N38150 X-5.476 
N38160 X-5.471 
N38170 X-5.465 
N38180 X-5.458 
N38190 X-5.451 
N38200 X-5.443 
N38210 X-5.434 
N38220 X-5.425 
N38230 X-5.416 
N38240 X-5.405 
N38250 X-5.394 
N38260 X-5.383 
N38270 X-5.371 
N38280 X-5.359 
N38290 X-5.346 
N38300 X-5.332 
N38310 X-5.318 
N38320 X-5.303 
N38330 X-5.288 
N38340 X-5.272 
N38350 X-5.256 
N38360 X-5.239 
N38370 X-5.222 
N38380 X-5.204 
N38390 X-5.186 
N38400 X-5.167 
N38410 X-5.147 
N38420 X-5.127 
N38430 X-5.107 
N38440 X-5.086 
N38450 X-5.065 
N38460 X-5.043 
N38470 X-5.021 
N38480 X-4.998 
N38490 X-4.975 
N38500 X-4.952 
N38510 X-4.928 
N38520 X-4.903 
N38530 X-4.878 
N38540 X-4.853 
N38550 X-4.827 
N38560 X-4.801 
N38570 X-4.774 
N38580 X-4.747 
N38590 X-4.72 
N38600 X-4.692 
N38610 X-4.664 
N38620 X-4.635 
N38630 X-4.606 
N38640 X-4.576 
N38650 X-4.547 
N38660 X-4.516 
N38670 X-4.486 
N38680 X-4.455 
N38690 X-4.424 
N38700 X-4.392 
N38710 X-4.36 
N38720 X-4.328 
N38730 X-4.295 
N38740 X-4.262 
N38750 X-4.228 
N38760 X-4.195 
N38770 X-4.161 
N38780 X-4.126 
N38790 X-4.092 
N38800 X-4.022 
N38810 X-3.95 
N38820 X-3.877 
N38830 X-3.804 
N38840 X-3.729 
N38850 X-3.653 
N38860 X-3.576 
N38870 X-3.498 
N38880 X-3.42 
N38890 X-3.34 
N38900 X-3.26 
N38910 X-3.178 
N38920 X-3.096 
N38930 X-3.013 
N38940 X-2.93 
N38950 X-2.846 
N38960 X-2.761 
N38970 X-2.675 
N38980 X-2.589 
N38990 X-2.503 
N39000 X-2.416 
N39010 X-2.329 
N39020 X-2.241 
N39030 X-2.153 
N39040 X-2.065 
N39050 X-1.887 
N39060 X-1.709 
N39070 X-1.351 
N39080 X-1.172 
N39090 X-0.993 
N39100 X-0.815 
N39110 X-0.639 
N39120 X-0.551 
N39130 X-0.463 
N39140 X-0.376 
N39150 X-0.289 
N39160 X-0.203 
N39170 X-0.118 
N39180 X-0.033 
N39190 X0.052 
N39200 X0.136 
N39210 X0.219 
N39220 X0.301 
N39230 X0.383 
N39240 X0.464 
N39250 X0.544 
N39260 X0.623 
N39270 X0.701 
N39280 X0.778 
N39290 X0.854 
N39300 X0.93 
N39310 X1.004 
N39320 X1.077 
N39330 X1.149 
N39340 X1.219 
N39350 X1.254 
N39360 X1.289 
N39370 X1.323 
N39380 X1.357 
N39390 X1.391 
N39400 X1.424 
N39410 X1.457 
N39420 X1.49 
N39430 X1.522 
N39440 X1.554 
N39450 X1.585 
N39460 X1.617 
N39470 X1.648 
N39480 X1.678 
N39490 X1.708 
N39500 X1.738 
N39510 X1.767 
N39520 X1.796 
N39530 X1.825 
N39540 X1.853 
N39550 X1.881 
N39560 X1.908 
N39570 X1.935 
N39580 X1.962 
N39590 X1.988 
N39600 X2.014 
N39610 X2.039 
N39620 X2.064 
N39630 X2.088 
N39640 X2.112 
N39650 X2.136 
N39660 X2.159 
N39670 X2.181 
N39680 X2.203 
N39690 X2.225 
N39700 X2.246 
N39710 X2.267 
N39720 X2.287 
N39730 X2.307 
N39740 X2.326 
N39750 X2.345 
N39760 X2.363 
N39770 X2.381 
N39780 X2.398 
N39790 X2.415 
N39800 X2.431 
N39810 X2.447 
N39820 X2.462 
N39830 X2.476 
N39840 X2.49 
N39850 X2.504 
N39860 X2.517 
N39870 X2.529 
N39880 X2.541 
N39890 X2.552 
N39900 X2.563 
N39910 X2.573 
N39920 X2.583 
N39930 X2.592 
N39940 X2.6 
N39950 X2.608 
N39960 X2.615 
N39970 X2.622 
N39980 X2.628 
N39990 X2.633 
N40000 X2.638 
N40010 X2.642 
N40020 X2.645 
N40030 X2.648 
N40040 X2.65 
N40050 X2.652 
N40060 X2.653 
N40070 X2.653 Y9.259 
N40080 X2.656 Y9.265 
N40090 X2.669 Y9.289 
N40100 X2.682 Y9.313 
N40110 X2.695 Y9.337 
N40120 X2.709 Y9.361 
N40130 X2.723 Y9.384 
N40140 X2.737 Y9.408 
N40150 X2.752 Y9.431 
N40160 X2.767 Y9.453 
N40170 X2.782 Y9.476 
N40180 X2.798 Y9.498 
N40190 X2.814 Y9.52 
N40200 X2.831 Y9.542 
N40210 X2.847 Y9.563 
N40220 X2.864 Y9.584 
N40230 X2.882 Y9.605 
N40240 X2.899 Y9.625 
N40250 X2.917 Y9.646 
N40260 X2.936 Y9.666 
N40270 X2.954 Y9.685 
N40280 X2.973 Y9.705 
N40290 X2.992 Y9.724 
N40300 X3.012 Y9.742 
N40310 X3.031 Y9.761 
N40320 X3.052 Y9.779 
N40330 X3.072 Y9.797 
N40340 X3.092 Y9.814 
N40350 X3.113 Y9.831 
N40360 X3.135 Y9.848 
N40370 X3.156 Y9.865 
N40380 X3.178 Y9.881 
N40390 X3.2 Y9.897 
N40400 X3.222 Y9.912 
N40410 X3.244 Y9.927 
N40420 X3.267 Y9.942 
N40430 X3.29 Y9.956 
N40440 X3.313 Y9.97 
N40450 X3.337 Y9.984 
N40460 X3.36 Y9.997 
N40470 X3.384 Y10.01 
N40480 X3.409 Y10.023 
N40490 X3.433 Y10.035 
N40500 X3.458 Y10.047 
N40510 X3.482 Y10.058 
N40520 X3.507 Y10.069 
N40530 X3.533 Y10.079 
N40540 X3.558 Y10.09 
N40550 X3.584 Y10.099 
N40560 X3.61 Y10.109 
N40570 X3.636 Y10.118 
N40580 X3.662 Y10.126 
N40590 X3.688 Y10.134 
N40600 X3.715 Y10.142 
N40610 X3.742 Y10.149 
N40620 X3.769 Y10.156 
N40630 X3.796 Y10.162 
N40640 X3.824 Y10.168 
N40650 X3.851 Y10.173 
N40660 X3.879 Y10.178 
N40670 X3.907 Y10.183 
N40680 X3.935 Y10.187 
N40690 X3.963 Y10.191 
N40700 X3.991 Y10.194 
N40710 X4.02 Y10.196 
N40720 X4.048 Y10.199 
N40730 X4.077 Y10.2 
N40740 X4.106 Y10.202 
N40750 X4.135 Y10.202 
N40760 X4.164 Y10.203 
N40770 Y10.202 
N40780 Y10.201 
N40790 Y10.199 
N40800 Y10.197 
N40810 Y10.196 
N40820 Y10.195 
N40830 X4.165 Y10.195 
N40840 X4.166 Y10.195 
N40850 X4.168 Y10.195 
N40860 X4.174 Y10.195 
N40870 X4.194 Y10.195 
N40880 X4.235 Y10.193 
N40890 X4.276 Y10.191 
N40900 X4.316 Y10.188 
N40910 X4.356 Y10.184 
N40920 X4.396 Y10.179 
N40930 X4.435 Y10.173 
N40940 X4.475 Y10.166 
N40950 X4.514 Y10.159 
N40960 X4.552 Y10.15 
N40970 X4.591 Y10.141 
N40980 X4.629 Y10.13 
N40990 X4.666 Y10.119 
N41000 X4.703 Y10.107 
N41010 X4.74 Y10.094 
N41020 X4.777 Y10.081 
N41030 X4.813 Y10.066 
N41040 X4.848 Y10.051 
N41050 X4.884 Y10.035 
N41060 X4.918 Y10.018 
N41070 X4.953 Y10 
N41080 X4.987 Y9.982 
N41090 X5.02 Y9.963 
N41100 X5.053 Y9.943 
N41110 X5.086 Y9.923 
N41120 X5.118 Y9.901 
N41130 X5.149 Y9.879 
N41140 X5.18 Y9.857 
N41150 X5.21 Y9.833 
N41160 X5.24 Y9.809 
N41170 X5.27 Y9.785 
N41180 X5.298 Y9.76 
N41190 X5.327 Y9.734 
N41200 X5.354 Y9.707 
N41210 X5.381 Y9.68 
N41220 X5.408 Y9.652 
N41230 X5.433 Y9.624 
N41240 X5.458 Y9.595 
N41250 X5.483 Y9.566 
N41260 X5.507 Y9.536 
N41270 X5.53 Y9.505 
N41280 X5.552 Y9.474 
N41290 X5.574 Y9.443 
N41300 X5.595 Y9.411 
N41310 X5.616 Y9.378 
N41320 X5.635 Y9.345 
N41330 X5.654 Y9.311 
N41340 X5.673 Y9.277 
N41350 X5.69 Y9.243 
N41360 X5.707 Y9.208 
N41370 X5.723 Y9.173 
N41380 X5.738 Y9.137 
N41390 X5.752 Y9.101 
N41400 X5.766 Y9.064 
N41410 X5.778 Y9.027 
N41420 X5.79 Y8.99 
N41430 X5.801 Y8.952 
N41440 X5.811 Y8.914 
N41450 X5.821 Y8.876 
N41460 X5.829 Y8.837 
N41470 X5.836 Y8.798 
N41480 X5.843 Y8.759 
N41490 X5.849 Y8.719 
N41500 X5.854 Y8.679 
N41510 X5.858 Y8.639 
N41520 X5.86 Y8.599 
N41530 X5.862 Y8.558 
N41540 X5.863 Y8.517 
N41550 X5.863 Y8.476 
N41560 X5.863 Y8.435 
N41570 X5.861 Y8.395 
N41580 X5.858 Y8.354 
N41590 X5.854 Y8.314 
N41600 X5.849 Y8.274 
N41610 X5.844 Y8.234 
N41620 X5.837 Y8.195 
N41630 X5.829 Y8.156 
N41640 X5.821 Y8.117 
N41650 X5.812 Y8.079 
N41660 X5.802 Y8.041 
N41670 X5.791 Y8.003 
N41680 X5.779 Y7.966 
N41690 X5.766 Y7.929 
N41700 X5.753 Y7.892 
N41710 X5.739 Y7.856 
N41720 X5.724 Y7.82 
N41730 X5.708 Y7.785 
N41740 X5.691 Y7.75 
N41750 X5.674 Y7.716 
N41760 X5.656 Y7.682 
N41770 X5.637 Y7.648 
N41780 X5.617 Y7.615 
N41790 X5.597 Y7.582 
N41800 X5.576 Y7.55 
N41810 X5.554 Y7.519 
N41820 X5.531 Y7.487 
N41830 X5.508 Y7.457 
N41840 X5.485 Y7.427 
N41850 X5.46 Y7.397 
N41860 X5.435 Y7.369 
N41870 X5.409 Y7.34 
N41880 X5.383 Y7.312 
N41890 X5.356 Y7.285 
N41900 X5.328 Y7.259 
N41910 X5.3 Y7.233 
N41920 X5.272 Y7.207 
N41930 X5.242 Y7.183 
N41940 X5.212 Y7.159 
N41950 X5.182 Y7.135 
N41960 X5.151 Y7.113 
N41970 X5.12 Y7.091 
N41980 X5.088 Y7.07 
N41990 X5.055 Y7.049 
N42000 X5.022 Y7.029 
N42010 X4.989 Y7.01 
N42020 X4.955 Y6.992 
N42030 X4.921 Y6.974 
N42040 X4.886 Y6.957 
N42050 X4.851 Y6.941 
N42060 X4.815 Y6.926 
N42070 X4.779 Y6.911 
N42080 X4.743 Y6.897 
N42090 X4.706 Y6.884 
N42100 X4.669 Y6.872 
N42110 X4.631 Y6.861 
N42120 X4.593 Y6.851 
N42130 X4.555 Y6.841 
N42140 X4.516 Y6.832 
N42150 X4.477 Y6.825 
N42160 X4.438 Y6.818 
N42170 X4.399 Y6.812 
N42180 X4.359 Y6.807 
N42190 X4.319 Y6.803 
N42200 X4.278 Y6.8 
N42210 X4.238 Y6.797 
N42220 X4.197 Y6.796 
N42230 X4.176 Y6.796 
N42240 X4.166 Y6.796 
N42250 X4.164 Y6.796 
N42260 X4.162 Y6.796 
N42270 X4.158 Y6.796 
N42280 X4.129 Y6.796 
N42290 X4.1 Y6.797 
N42300 X4.071 Y6.798 
N42310 X4.042 Y6.8 
N42320 X4.014 Y6.802 
N42330 X3.985 Y6.805 
N42340 X3.957 Y6.808 
N42350 X3.929 Y6.812 
N42360 X3.901 Y6.816 
N42370 X3.873 Y6.821 
N42380 X3.846 Y6.826 
N42390 X3.818 Y6.831 
N42400 X3.791 Y6.837 
N42410 X3.764 Y6.844 
N42420 X3.737 Y6.851 
N42430 X3.71 Y6.858 
N42440 X3.683 Y6.866 
N42450 X3.657 Y6.874 
N42460 X3.631 Y6.882 
N42470 X3.605 Y6.891 
N42480 X3.579 Y6.901 
N42490 X3.553 Y6.911 
N42500 X3.528 Y6.921 
N42510 X3.502 Y6.932 
N42520 X3.477 Y6.943 
N42530 X3.453 Y6.954 
N42540 X3.428 Y6.966 
N42550 X3.404 Y6.978 
N42560 X3.38 Y6.991 
N42570 X3.356 Y7.004 
N42580 X3.332 Y7.017 
N42590 X3.309 Y7.031 
N42600 X3.285 Y7.045 
N42610 X3.263 Y7.059 
N42620 X3.24 Y7.074 
N42630 X3.217 Y7.089 
N42640 X3.195 Y7.105 
N42650 X3.173 Y7.121 
N42660 X3.152 Y7.137 
N42670 X3.13 Y7.153 
N42680 X3.109 Y7.17 
N42690 X3.088 Y7.187 
N42700 X3.068 Y7.205 
N42710 X3.047 Y7.223 
N42720 X3.027 Y7.241 
N42730 X3.008 Y7.259 
N42740 X2.988 Y7.278 
N42750 X2.969 Y7.297 
N42760 X2.95 Y7.317 
N42770 X2.932 Y7.337 
N42780 X2.914 Y7.357 
N42790 X2.896 Y7.377 
N42800 X2.878 Y7.397 
N42810 X2.861 Y7.418 
N42820 X2.844 Y7.44 
N42830 X2.827 Y7.461 
N42840 X2.811 Y7.483 
N42850 X2.795 Y7.505 
N42860 X2.779 Y7.527 
N42870 X2.764 Y7.549 
N42880 X2.749 Y7.572 
N42890 X2.734 Y7.595 
N42900 X2.72 Y7.618 
N42910 X2.706 Y7.642 
N42920 X2.693 Y7.666 
N42930 X2.679 Y7.69 
N42940 X2.666 Y7.714 
N42950 X2.654 Y7.738 
N42960 X2.653 Y7.74 
N42970 X2.652 Y7.74 
N42980 X2.651 
N42990 X2.649 
N43000 X2.646 
N43010 X2.643 
N43020 X2.64 
N43030 X2.635 
N43040 X2.631 
N43050 X2.625 
N43060 X2.619 
N43070 X2.613 
N43080 X2.606 
N43090 X2.598 
N43100 X2.59 
N43110 X2.581 
N43120 X2.572 
N43130 X2.562 
N43140 X2.552 
N43150 X2.541 
N43160 X2.53 
N43170 X2.518 
N43180 X2.505 
N43190 X2.493 
N43200 X2.479 
N43210 X2.465 
N43220 X2.451 
N43230 X2.436 
N43240 X2.421 
N43250 X2.405 
N43260 X2.389 
N43270 X2.372 
N43280 X2.355 
N43290 X2.337 
N43300 X2.319 
N43310 X2.3 
N43320 X2.281 
N43330 X2.262 
N43340 X2.242 
N43350 X2.222 
N43360 X2.201 
N43370 X2.18 
N43380 X2.158 
N43390 X2.136 
N43400 X2.114 
N43410 X2.091 
N43420 X2.067 
N43430 X2.044 
N43440 X2.02 
N43450 X1.995 
N43460 X1.971 
N43470 X1.945 
N43480 X1.92 
N43490 X1.894 
N43500 X1.867 
N43510 X1.841 
N43520 X1.814 
N43530 X1.786 
N43540 X1.759 
N43550 X1.731 
N43560 X1.702 
N43570 X1.673 
N43580 X1.644 
N43590 X1.615 
N43600 X1.585 
N43610 X1.555 
N43620 X1.494 
N43630 X1.432 
N43640 X1.368 
N43650 X1.304 
N43660 X1.238 
N43670 X1.171 
N43680 X1.103 
N43690 X1.034 
N43700 X0.965 
N43710 X0.894 
N43720 X0.822 
N43730 X0.75 
N43740 X0.676 
N43750 X0.602 
N43760 X0.527 
N43770 X0.452 
N43780 X0.375 
N43790 X0.298 
N43800 X0.221 
N43810 X0.143 
N43820 X0.064 
N43830 X-0.015 
N43840 X-0.095 
N43850 X-0.175 
N43860 X-0.256 
N43870 X-0.337 
N43880 X-0.418 
N43890 X-0.581 
N43900 X-0.746 
N43910 X-0.91 
N43920 X-1.241 
N43930 X-1.406 
N43940 X-1.571 
N43950 X-1.734 
N43960 X-1.897 
N43970 X-1.978 
N43980 X-2.058 
N43990 X-2.138 
N44000 X-2.218 
N44010 X-2.297 
N44020 X-2.376 
N44030 X-2.454 
N44040 X-2.531 
N44050 X-2.608 
N44060 X-2.684 
N44070 X-2.76 
N44080 X-2.835 
N44090 X-2.909 
N44100 X-2.982 
N44110 X-3.054 
N44120 X-3.126 
N44130 X-3.196 
N44140 X-3.266 
N44150 X-3.334 
N44160 X-3.402 
N44170 X-3.469 
N44180 X-3.534 
N44190 X-3.599 
N44200 X-3.662 
N44210 X-3.724 
N44220 X-3.754 
N44230 X-3.785 
N44240 X-3.815 
N44250 X-3.844 
N44260 X-3.873 
N44270 X-3.902 
N44280 X-3.931 
N44290 X-3.959 
N44300 X-3.987 
N44310 X-4.015 
N44320 X-4.042 
N44330 X-4.069 
N44340 X-4.095 
N44350 X-4.122 
N44360 X-4.147 
N44370 X-4.173 
N44380 X-4.198 
N44390 X-4.223 
N44400 X-4.247 
N44410 X-4.271 
N44420 X-4.294 
N44430 X-4.317 
N44440 X-4.34 
N44450 X-4.362 
N44460 X-4.384 
N44470 X-4.406 
N44480 X-4.427 
N44490 X-4.447 
N44500 X-4.467 
N44510 X-4.487 
N44520 X-4.506 
N44530 X-4.525 
N44540 X-4.544 
N44550 X-4.562 
N44560 X-4.579 
N44570 X-4.596 
N44580 X-4.613 
N44590 X-4.629 
N44600 X-4.644 
N44610 X-4.66 
N44620 X-4.674 
N44630 X-4.688 
N44640 X-4.702 
N44650 X-4.715 
N44660 X-4.728 
N44670 X-4.74 
N44680 X-4.752 
N44690 X-4.763 
N44700 X-4.773 
N44710 X-4.783 
N44720 X-4.793 
N44730 X-4.802 
N44740 X-4.811 
N44750 X-4.819 
N44760 X-4.826 
N44770 X-4.833 
N44780 X-4.839 
N44790 X-4.845 
N44800 X-4.85 
N44810 X-4.855 
N44820 X-4.859 
N44830 X-4.862 
N44840 X-4.865 
N44850 X-4.867 
N44860 X-4.869 
N44870 X-4.87 
N44880 X-4.871 
N44890 X-4.871 Y7.739 
N44900 X-4.873 Y7.738 
N44910 X-4.875 Y7.736 
N44920 X-4.877 Y7.733 
N44930 X-4.881 Y7.73 
N44940 X-4.885 Y7.726 
N44950 X-4.89 Y7.721 
N44960 X-4.895 Y7.715 
N44970 X-4.901 Y7.709 
N44980 X-4.908 Y7.703 
N44990 X-4.915 Y7.695 
N45000 X-4.923 Y7.687 
N45010 X-4.932 Y7.679 
N45020 X-4.941 Y7.67 
N45030 X-4.951 Y7.66 
N45040 X-4.961 Y7.65 
N45050 X-4.972 Y7.639 
N45060 X-4.984 Y7.627 
N45070 X-4.996 Y7.615 
N45080 X-5.008 Y7.603 
N45090 X-5.021 Y7.59 
N45100 X-5.035 Y7.576 
N45110 X-5.049 Y7.562 
N45120 X-5.063 Y7.548 
N45130 X-5.078 Y7.533 
N45140 X-5.094 Y7.517 
N45150 X-5.11 Y7.501 
N45160 X-5.126 Y7.485 
N45170 X-5.143 Y7.468 
N45180 X-5.16 Y7.451 
N45190 X-5.178 Y7.434 
N45200 X-5.196 Y7.416 
N45210 X-5.214 Y7.397 
N45220 X-5.233 Y7.379 
N45230 X-5.252 Y7.359 
N45240 X-5.272 Y7.34 
N45250 X-5.292 Y7.32 
N45260 X-5.312 Y7.3 
N45270 X-5.333 Y7.28 
N45280 X-5.353 Y7.259 
N45290 X-5.375 Y7.238 
N45300 X-5.396 Y7.216 
N45310 X-5.418 Y7.195 
N45320 X-5.44 Y7.173 
N45330 X-5.462 Y7.151 
N45340 X-5.484 Y7.128 
N45350 X-5.507 Y7.105 
N45360 X-5.553 Y7.059 
N45370 X-5.6 Y7.013 
N45380 X-5.648 Y6.965 
N45390 X-5.696 Y6.917 
N45400 X-5.745 Y6.868 
N45410 X-5.795 Y6.819 
N45420 X-5.844 Y6.769 
N45430 X-5.945 Y6.669 
N45440 X-6.046 Y6.569 
N45450 X-6.146 Y6.468 
N45460 X-6.196 Y6.418 
N45470 X-6.246 Y6.369 
N45480 X-6.296 Y6.32 
N45490 X-6.344 Y6.271 
N45500 X-6.393 Y6.223 
N45510 X-6.44 Y6.175 
N45520 X-6.487 Y6.129 
N45530 X-6.533 Y6.083 
N45540 X-6.556 Y6.06 
N45550 X-6.579 Y6.038 
N45560 X-6.601 Y6.015 
N45570 X-6.623 Y5.994 
N45580 X-6.644 Y5.972 
N45590 X-6.666 Y5.951 
N45600 X-6.687 Y5.93 
N45610 X-6.708 Y5.909 
N45620 X-6.728 Y5.888 
N45630 X-6.748 Y5.868 
N45640 X-6.768 Y5.848 
N45650 X-6.788 Y5.829 
N45660 X-6.807 Y5.81 
N45670 X-6.826 Y5.791 
N45680 X-6.844 Y5.773 
N45690 X-6.862 Y5.755 
N45700 X-6.88 Y5.738 
N45710 X-6.897 Y5.72 
N45720 X-6.914 Y5.704 
N45730 X-6.93 Y5.687 
N45740 X-6.946 Y5.672 
N45750 X-6.961 Y5.656 
N45760 X-6.976 Y5.641 
N45770 X-6.991 Y5.627 
N45780 X-7.005 Y5.613 
N45790 X-7.018 Y5.6 
N45800 X-7.031 Y5.587 
N45810 X-7.044 Y5.574 
N45820 X-7.055 Y5.562 
N45830 X-7.067 Y5.551 
N45840 X-7.078 Y5.54 
N45850 X-7.088 Y5.53 
N45860 X-7.098 Y5.52 
N45870 X-7.107 Y5.511 
N45880 X-7.115 Y5.503 
N45890 X-7.123 Y5.495 
N45900 X-7.13 Y5.488 
N45910 X-7.137 Y5.481 
N45920 X-7.143 Y5.475 
N45930 X-7.148 Y5.47 
N45940 X-7.153 Y5.465 
N45950 X-7.157 Y5.461 
N45960 X-7.161 Y5.457 
N45970 X-7.163 Y5.455 
N45980 X-7.165 Y5.453 
N45990 X-7.166 Y5.452 
N46000 X-7.167 Y5.451 
N46010 X-7.167 Y5.45 
N46020 Y5.448 
N46030 Y5.447 
N46040 Y5.445 
N46050 Y5.443 
N46060 Y5.44 
N46070 Y5.437 
N46080 Y5.434 
N46090 Y5.43 
N46100 Y5.426 
N46110 Y5.422 
N46120 Y5.412 
N46130 Y5.401 
N46140 Y5.389 
N46150 Y5.376 
N46160 Y5.362 
N46170 Y5.347 
N46180 Y5.331 
N46190 Y5.314 
N46200 Y5.296 
N46210 Y5.278 
N46220 Y5.258 
N46230 Y5.238 
N46240 Y5.217 
N46250 Y5.195 
N46260 Y5.173 
N46270 Y5.15 
N46280 Y5.127 
N46290 Y5.103 
N46300 Y5.078 
N46310 Y5.054 
N46320 Y5.003 
N46330 Y4.952 
N46340 Y4.9 
N46350 Y4.847 
N46360 Y4.795 
N46370 Y4.743 
N46380 Y4.692 
N46390 Y4.667 
N46400 Y4.642 
N46410 Y4.617 
N46420 Y4.593 
N46430 Y4.57 
N46440 Y4.546 
N46450 Y4.524 
N46460 Y4.502 
N46470 Y4.481 
N46480 Y4.46 
N46490 Y4.44 
N46500 Y4.421 
N46510 Y4.403 
N46520 Y4.385 
N46530 Y4.369 
N46540 Y4.353 
N46550 Y4.339 
N46560 Y4.325 
N46570 Y4.313 
N46580 Y4.301 
N46590 Y4.291 
N46600 Y4.287 
N46610 Y4.283 
N46620 Y4.279 
N46630 Y4.275 
N46640 Y4.272 
N46650 Y4.269 
N46660 Y4.266 
N46670 Y4.264 
N46680 Y4.262 
N46690 Y4.26 
N46700 Y4.259 
N46710 Y4.258 
N46720 X-7.167 Y4.257 
N46730 X-7.164 Y4.256 
N46740 X-7.139 Y4.243 
N46750 X-7.115 Y4.231 
N46760 X-7.091 Y4.217 
N46770 X-7.067 Y4.204 
N46780 X-7.044 Y4.19 
N46790 X-7.021 Y4.175 
N46800 X-6.998 Y4.161 
N46810 X-6.975 Y4.146 
N46820 X-6.952 Y4.13 
N46830 X-6.93 Y4.115 
N46840 X-6.908 Y4.099 
N46850 X-6.887 Y4.082 
N46860 X-6.865 Y4.066 
N46870 X-6.844 Y4.049 
N46880 X-6.823 Y4.031 
N46890 X-6.803 Y4.014 
N46900 X-6.782 Y3.996 
N46910 X-6.762 Y3.978 
N46920 X-6.743 Y3.959 
N46930 X-6.723 Y3.94 
N46940 X-6.704 Y3.921 
N46950 X-6.685 Y3.902 
N46960 X-6.667 Y3.882 
N46970 X-6.649 Y3.862 
N46980 X-6.631 Y3.842 
N46990 X-6.613 Y3.821 
N47000 X-6.596 Y3.8 
N47010 X-6.579 Y3.779 
N47020 X-6.563 Y3.758 
N47030 X-6.546 Y3.736 
N47040 X-6.531 Y3.714 
N47050 X-6.515 Y3.692 
N47060 X-6.5 Y3.669 
N47070 X-6.485 Y3.647 
N47080 X-6.471 Y3.624 
N47090 X-6.457 Y3.601 
N47100 X-6.443 Y3.577 
N47110 X-6.43 Y3.553 
N47120 X-6.417 Y3.53 
N47130 X-6.404 Y3.505 
N47140 X-6.392 Y3.481 
N47150 X-6.38 Y3.456 
N47160 X-6.369 Y3.432 
N47170 X-6.358 Y3.407 
N47180 X-6.347 Y3.381 
N47190 X-6.337 Y3.356 
N47200 X-6.327 Y3.33 
N47210 X-6.318 Y3.304 
N47220 X-6.309 Y3.278 
N47230 X-6.3 Y3.252 
N47240 X-6.292 Y3.226 
N47250 X-6.284 Y3.199 
N47260 X-6.277 Y3.172 
N47270 X-6.27 Y3.145 
N47280 X-6.264 Y3.118 
N47290 X-6.258 Y3.091 
N47300 X-6.253 Y3.063 
N47310 X-6.248 Y3.036 
N47320 X-6.243 Y3.008 
N47330 X-6.239 Y2.98 
N47340 X-6.235 Y2.952 
N47350 X-6.232 Y2.923 
N47360 X-6.229 Y2.895 
N47370 X-6.227 Y2.866 
N47380 X-6.225 Y2.838 
N47390 X-6.224 Y2.809 
N47400 X-6.223 Y2.78 
N47410 X-6.223 Y2.751 
N47420 X-6.223 Y2.747 
N47430 X-6.223 Y2.742 
N47440 X-6.223 Y2.732 
N47450 X-6.223 Y2.711 
N47460 X-6.224 Y2.67 
N47470 X-6.227 Y2.63 
N47480 X-6.23 Y2.589 
N47490 X-6.234 Y2.549 
N47500 X-6.239 Y2.51 
N47510 X-6.245 Y2.47 
N47520 X-6.252 Y2.431 
N47530 G00 Z5 
N47540 G00 X-9.416 Y8.275 
N47550 G01 Z-5 F254 
N47560 G01 X-9.463 Y8.25 F1200 
N47570 X-9.512 Y8.226 
N47580 X-9.561 Y8.204 
N47590 X-9.611 Y8.183 
N47600 X-9.662 Y8.164 
N47610 X-9.714 Y8.146 
N47620 X-9.767 Y8.13 
N47630 X-9.82 Y8.116 
N47640 X-9.874 Y8.103 
N47650 X-9.928 Y8.092 
N47660 X-9.983 Y8.083 
N47670 X-10.039 Y8.076 
N47680 X-10.095 Y8.07 
N47690 X-10.152 Y8.067 
N47700 X-10.209 Y8.065 
N47710 X-10.267 Y8.065 
N47720 X-10.324 Y8.067 
N47730 X-10.381 Y8.071 
N47740 X-10.437 Y8.077 
N47750 X-10.492 Y8.084 
N47760 X-10.547 Y8.094 
N47770 X-10.602 Y8.105 
N47780 X-10.655 Y8.118 
N47790 X-10.709 Y8.132 
N47800 X-10.761 Y8.148 
N47810 X-10.813 Y8.166 
N47820 X-10.863 Y8.186 
N47830 X-10.914 Y8.207 
N47840 X-10.963 Y8.229 
N47850 X-11.011 Y8.253 
N47860 X-11.059 Y8.279 
N47870 X-11.106 Y8.306 
N47880 X-11.151 Y8.334 
N47890 X-11.196 Y8.364 
N47900 X-11.24 Y8.395 
N47910 X-11.282 Y8.428 
N47920 X-11.324 Y8.462 
N47930 X-11.364 Y8.497 
N47940 X-11.404 Y8.533 
N47950 X-11.442 Y8.571 
N47960 X-11.479 Y8.609 
N47970 X-11.515 Y8.649 
N47980 X-11.55 Y8.69 
N47990 X-11.583 Y8.732 
N48000 X-11.615 Y8.775 
N48010 X-11.646 Y8.819 
N48020 X-11.675 Y8.864 
N48030 X-11.703 Y8.91 
N48040 X-11.729 Y8.957 
N48050 X-11.754 Y9.005 
N48060 X-11.778 Y9.054 
N48070 X-11.8 Y9.104 
N48080 X-11.82 Y9.154 
N48090 X-11.839 Y9.205 
N48100 X-11.856 Y9.257 
N48110 X-11.872 Y9.31 
N48120 X-11.886 Y9.363 
N48130 X-11.898 Y9.417 
N48140 X-11.908 Y9.472 
N48150 X-11.917 Y9.527 
N48160 X-11.924 Y9.583 
N48170 X-11.929 Y9.639 
N48180 X-11.932 Y9.696 
N48190 X-11.933 Y9.753 
N48200 X-11.933 Y9.811 
N48210 X-11.93 Y9.868 
N48220 X-11.926 Y9.924 
N48230 X-11.92 Y9.98 
N48240 X-11.912 Y10.036 
N48250 X-11.902 Y10.091 
N48260 X-11.89 Y10.145 
N48270 X-11.877 Y10.199 
N48280 X-11.862 Y10.252 
N48290 X-11.846 Y10.304 
N48300 X-11.827 Y10.355 
N48310 X-11.808 Y10.406 
N48320 X-11.786 Y10.456 
N48330 X-11.763 Y10.505 
N48340 X-11.739 Y10.553 
N48350 X-11.713 Y10.601 
N48360 X-11.686 Y10.647 
N48370 X-11.657 Y10.692 
N48380 X-11.627 Y10.737 
N48390 X-11.595 Y10.78 
N48400 X-11.562 Y10.823 
N48410 X-11.528 Y10.864 
N48420 X-11.493 Y10.905 
N48430 X-11.456 Y10.944 
N48440 X-11.419 Y10.982 
N48450 X-11.38 Y11.018 
N48460 X-11.34 Y11.054 
N48470 X-11.298 Y11.088 
N48480 X-11.256 Y11.121 
N48490 X-11.213 Y11.153 
N48500 X-11.168 Y11.183 
N48510 X-11.123 Y11.212 
N48520 X-11.077 Y11.24 
N48530 X-11.03 Y11.266 
N48540 X-10.981 Y11.29 
N48550 X-10.932 Y11.314 
N48560 X-10.883 Y11.335 
N48570 X-10.832 Y11.355 
N48580 X-10.781 Y11.374 
N48590 X-10.729 Y11.391 
N48600 X-10.676 Y11.406 
N48610 X-10.622 Y11.419 
N48620 X-10.568 Y11.431 
N48630 X-10.513 Y11.441 
N48640 X-10.458 Y11.449 
N48650 X-10.402 Y11.456 
N48660 X-10.346 Y11.46 
N48670 X-10.289 Y11.463 
N48680 X-10.26 Y11.464 
N48690 X-10.246 Y11.464 
N48700 X-10.238 Y11.464 
N48710 X-10.235 Y11.464 
N48720 X-10.234 
N48730 X-10.233 
N48740 X-10.222 Y11.464 
N48750 X-10.199 Y11.464 
N48760 X-10.152 Y11.461 
N48770 X-10.107 Y11.457 
N48780 X-10.061 Y11.452 
N48790 X-10.016 Y11.446 
N48800 X-9.972 Y11.438 
N48810 X-9.928 Y11.429 
N48820 X-9.884 Y11.419 
N48830 X-9.841 Y11.408 
N48840 X-9.799 Y11.396 
N48850 X-9.757 Y11.384 
N48860 X-9.715 Y11.371 
N48870 X-9.705 Y11.368 
N48880 X-9.7 Y11.367 
N48890 X-9.698 Y11.366 
N48900 X-9.697 Y11.366 
N48910 X-9.697 Y11.367 
N48920 X-9.696 Y11.368 
N48930 X-9.694 Y11.369 
N48940 X-9.692 Y11.371 
N48950 X-9.69 Y11.373 
N48960 X-9.687 Y11.376 
N48970 X-9.684 Y11.379 
N48980 X-9.681 Y11.383 
N48990 X-9.673 Y11.39 
N49000 X-9.664 Y11.4 
N49010 X-9.653 Y11.411 
N49020 X-9.641 Y11.423 
N49030 X-9.627 Y11.436 
N49040 X-9.612 Y11.451 
N49050 X-9.596 Y11.467 
N49060 X-9.578 Y11.485 
N49070 X-9.56 Y11.504 
N49080 X-9.54 Y11.523 
N49090 X-9.519 Y11.544 
N49100 X-9.497 Y11.567 
N49110 X-9.474 Y11.59 
N49120 X-9.449 Y11.614 
N49130 X-9.424 Y11.639 
N49140 X-9.398 Y11.666 
N49150 X-9.37 Y11.693 
N49160 X-9.342 Y11.721 
N49170 X-9.313 Y11.75 
N49180 X-9.283 Y11.78 
N49190 X-9.253 Y11.811 
N49200 X-9.221 Y11.842 
N49210 X-9.189 Y11.874 
N49220 X-9.156 Y11.907 
N49230 X-9.122 Y11.941 
N49240 X-9.088 Y11.975 
N49250 X-9.053 Y12.01 
N49260 X-9.018 Y12.046 
N49270 X-8.982 Y12.082 
N49280 X-8.945 Y12.118 
N49290 X-8.908 Y12.155 
N49300 X-8.871 Y12.193 
N49310 X-8.833 Y12.231 
N49320 X-8.794 Y12.269 
N49330 X-8.717 Y12.346 
N49340 X-8.638 Y12.425 
N49350 X-8.559 Y12.505 
N49360 X-8.238 Y12.825 
N49370 X-8.158 Y12.905 
N49380 X-8.079 Y12.984 
N49390 X-8.002 Y13.062 
N49400 X-7.925 Y13.138 
N49410 X-7.888 Y13.176 
N49420 X-7.85 Y13.213 
N49430 X-7.814 Y13.25 
N49440 X-7.777 Y13.286 
N49450 X-7.742 Y13.322 
N49460 X-7.707 Y13.357 
N49470 X-7.672 Y13.391 
N49480 X-7.638 Y13.425 
N49490 X-7.605 Y13.458 
N49500 X-7.572 Y13.491 
N49510 X-7.541 Y13.523 
N49520 X-7.51 Y13.554 
N49530 X-7.479 Y13.584 
N49540 X-7.45 Y13.613 
N49550 X-7.422 Y13.642 
N49560 X-7.394 Y13.669 
N49570 X-7.367 Y13.696 
N49580 X-7.342 Y13.722 
N49590 X-7.317 Y13.746 
N49600 X-7.293 Y13.77 
N49610 X-7.271 Y13.793 
N49620 X-7.249 Y13.814 
N49630 X-7.229 Y13.834 
N49640 X-7.21 Y13.853 
N49650 X-7.192 Y13.871 
N49660 X-7.175 Y13.888 
N49670 X-7.16 Y13.903 
N49680 X-7.146 Y13.917 
N49690 X-7.133 Y13.93 
N49700 X-7.122 Y13.942 
N49710 X-7.112 Y13.951 
N49720 X-7.103 Y13.96 
N49730 X-7.1 Y13.964 
N49740 X-7.096 Y13.967 
N49750 X-7.093 Y13.97 
N49760 X-7.091 Y13.972 
N49770 X-7.089 Y13.975 
N49780 X-7.087 Y13.976 
N49790 X-7.086 Y13.978 
N49800 X-7.085 Y13.979 
N49810 X-7.084 Y13.979 
N49820 X-7.083 Y13.979 
N49830 X-7.082 
N49840 X-7.081 
N49850 X-7.078 
N49860 X-7.075 
N49870 X-7.072 
N49880 X-7.068 
N49890 X-7.063 
N49900 X-7.057 
N49910 X-7.051 
N49920 X-7.045 
N49930 X-7.038 
N49940 X-7.03 
N49950 X-7.021 
N49960 X-7.012 
N49970 X-7.003 
N49980 X-6.993 
N49990 X-6.982 
N50000 X-6.971 
N50010 X-6.959 
N50020 X-6.946 
N50030 X-6.933 
N50040 X-6.92 
N50050 X-6.906 
N50060 X-6.891 
N50070 X-6.876 
N50080 X-6.86 
N50090 X-6.844 
N50100 X-6.827 
N50110 X-6.809 
N50120 X-6.791 
N50130 X-6.773 
N50140 X-6.754 
N50150 X-6.734 
N50160 X-6.694 
N50170 X-6.651 
N50180 X-6.606 
N50190 X-6.559 
N50200 X-6.51 
N50210 X-6.46 
N50220 X-6.407 
N50230 X-6.352 
N50240 X-6.296 
N50250 X-6.237 
N50260 X-6.177 
N50270 X-6.115 
N50280 X-6.051 
N50290 X-5.986 
N50300 X-5.919 
N50310 X-5.85 
N50320 X-5.779 
N50330 X-5.707 
N50340 X-5.633 
N50350 X-5.557 
N50360 X-5.48 
N50370 X-5.401 
N50380 X-5.321 
N50390 X-5.239 
N50400 X-5.156 
N50410 X-5.072 
N50420 X-4.986 
N50430 X-4.898 
N50440 X-4.81 
N50450 X-4.719 
N50460 X-4.628 
N50470 X-4.535 
N50480 X-4.441 
N50490 X-4.346 
N50500 X-4.25 
N50510 X-4.152 
N50520 X-4.053 
N50530 X-3.953 
N50540 X-3.852 
N50550 X-3.75 
N50560 X-3.647 
N50570 X-3.543 
N50580 X-3.438 
N50590 X-3.332 
N50600 X-3.225 
N50610 X-3.117 
N50620 X-3.008 
N50630 X-2.898 
N50640 X-2.787 
N50650 X-2.676 
N50660 X-2.563 
N50670 X-2.45 
N50680 X-2.337 
N50690 X-2.222 
N50700 X-2.107 
N50710 X-1.991 
N50720 X-1.875 
N50730 X-1.758 
N50740 X-1.64 
N50750 X-1.522 
N50760 X-1.403 
N50770 X-1.164 
N50780 X-0.923 
N50790 X-0.681 
N50800 X-0.437 
N50810 X-0.192 
N50820 X0.054 
N50830 X0.3 
N50840 X0.548 
N50850 X1.538 
N50860 X1.785 
N50870 X2.032 
N50880 X2.277 
N50890 X2.522 
N50900 X2.765 
N50910 X3.006 
N50920 X3.246 
N50930 X3.484 
N50940 X3.602 
N50950 X3.719 
N50960 X3.836 
N50970 X3.953 
N50980 X4.068 
N50990 X4.183 
N51000 X4.298 
N51010 X4.411 
N51020 X4.524 
N51030 X4.636 
N51040 X4.748 
N51050 X4.858 
N51060 X4.968 
N51070 X5.077 
N51080 X5.185 
N51090 X5.292 
N51100 X5.398 
N51110 X5.503 
N51120 X5.607 
N51130 X5.71 
N51140 X5.812 
N51150 X5.912 
N51160 X6.012 
N51170 X6.111 
N51180 X6.208 
N51190 X6.304 
N51200 X6.4 
N51210 X6.493 
N51220 X6.586 
N51230 X6.677 
N51240 X6.767 
N51250 X6.856 
N51260 X6.943 
N51270 X7.029 
N51280 X7.113 
N51290 X7.196 
N51300 X7.278 
N51310 X7.357 
N51320 X7.436 
N51330 X7.513 
N51340 X7.588 
N51350 X7.662 
N51360 X7.734 
N51370 X7.804 
N51380 X7.873 
N51390 X7.94 
N51400 X8.005 
N51410 X8.069 
N51420 X8.131 
N51430 X8.191 
N51440 X8.249 
N51450 X8.305 
N51460 X8.359 
N51470 X8.412 
N51480 X8.462 
N51490 X8.511 
N51500 X8.557 
N51510 X8.602 
N51520 X8.644 
N51530 X8.685 
N51540 X8.704 
N51550 X8.723 
N51560 X8.741 
N51570 X8.759 
N51580 X8.776 
N51590 X8.793 
N51600 X8.809 
N51610 X8.825 
N51620 X8.84 
N51630 X8.855 
N51640 X8.869 
N51650 X8.882 
N51660 X8.895 
N51670 X8.907 
N51680 X8.919 
N51690 X8.93 
N51700 X8.941 
N51710 X8.95 
N51720 X8.96 
N51730 X8.969 
N51740 X8.977 
N51750 X8.985 
N51760 X8.992 
N51770 X8.998 
N51780 X9.004 
N51790 X9.009 
N51800 X9.014 
N51810 X9.018 
N51820 X9.021 
N51830 X9.024 
N51840 X9.026 
N51850 X9.028 
N51860 X9.029 Y13.979 
N51870 X9.03 Y13.978 
N51880 X9.032 Y13.976 
N51890 X9.035 Y13.973 
N51900 X9.039 Y13.969 
N51910 X9.043 Y13.965 
N51920 X9.048 Y13.96 
N51930 X9.054 Y13.954 
N51940 X9.061 Y13.947 
N51950 X9.068 Y13.94 
N51960 X9.077 Y13.932 
N51970 X9.085 Y13.923 
N51980 X9.095 Y13.913 
N51990 X9.105 Y13.903 
N52000 X9.116 Y13.892 
N52010 X9.128 Y13.88 
N52020 X9.14 Y13.868 
N52030 X9.153 Y13.855 
N52040 X9.167 Y13.841 
N52050 X9.181 Y13.827 
N52060 X9.196 Y13.812 
N52070 X9.212 Y13.796 
N52080 X9.228 Y13.78 
N52090 X9.245 Y13.763 
N52100 X9.263 Y13.745 
N52110 X9.281 Y13.727 
N52120 X9.3 Y13.709 
N52130 X9.319 Y13.689 
N52140 X9.339 Y13.669 
N52150 X9.359 Y13.649 
N52160 X9.38 Y13.628 
N52170 X9.402 Y13.606 
N52180 X9.424 Y13.584 
N52190 X9.447 Y13.562 
N52200 X9.47 Y13.538 
N52210 X9.494 Y13.515 
N52220 X9.518 Y13.49 
N52230 X9.543 Y13.466 
N52240 X9.568 Y13.44 
N52250 X9.593 Y13.415 
N52260 X9.62 Y13.388 
N52270 X9.646 Y13.362 
N52280 X9.674 Y13.335 
N52290 X9.701 Y13.307 
N52300 X9.729 Y13.279 
N52310 X9.758 Y13.25 
N52320 X9.787 Y13.222 
N52330 X9.816 Y13.192 
N52340 X9.846 Y13.162 
N52350 X9.876 Y13.132 
N52360 X9.906 Y13.102 
N52370 X9.937 Y13.071 
N52380 X9.969 Y13.039 
N52390 X10.032 Y12.976 
N52400 X10.098 Y12.91 
N52410 X10.164 Y12.844 
N52420 X10.232 Y12.776 
N52430 X10.301 Y12.707 
N52440 X10.371 Y12.637 
N52450 X10.443 Y12.566 
N52460 X10.515 Y12.493 
N52470 X10.588 Y12.42 
N52480 X10.662 Y12.346 
N52490 X10.737 Y12.271 
N52500 X10.813 Y12.195 
N52510 X10.889 Y12.119 
N52520 X10.966 Y12.042 
N52530 X11.044 Y11.964 
N52540 X11.122 Y11.886 
N52550 X11.201 Y11.808 
N52560 X11.359 Y11.65 
N52570 X11.677 Y11.332 
N52580 X11.835 Y11.173 
N52590 X11.994 Y11.014 
N52600 X12.072 Y10.936 
N52610 X12.151 Y10.858 
N52620 X12.228 Y10.78 
N52630 X12.306 Y10.702 
N52640 X12.382 Y10.626 
N52650 X12.458 Y10.55 
N52660 X12.534 Y10.474 
N52670 X12.608 Y10.4 
N52680 X12.682 Y10.326 
N52690 X12.755 Y10.253 
N52700 X12.827 Y10.182 
N52710 X12.897 Y10.111 
N52720 X12.967 Y10.041 
N52730 X13.035 Y9.973 
N52740 X13.103 Y9.906 
N52750 X13.168 Y9.84 
N52760 X13.233 Y9.775 
N52770 X13.265 Y9.744 
N52780 X13.296 Y9.712 
N52790 X13.327 Y9.681 
N52800 X13.357 Y9.651 
N52810 X13.387 Y9.621 
N52820 X13.417 Y9.591 
N52830 X13.447 Y9.562 
N52840 X13.475 Y9.533 
N52850 X13.504 Y9.504 
N52860 X13.532 Y9.476 
N52870 X13.56 Y9.449 
N52880 X13.587 Y9.421 
N52890 X13.613 Y9.395 
N52900 X13.639 Y9.369 
N52910 X13.665 Y9.343 
N52920 X13.69 Y9.318 
N52930 X13.715 Y9.293 
N52940 X13.739 Y9.269 
N52950 X13.763 Y9.245 
N52960 X13.786 Y9.222 
N52970 X13.809 Y9.199 
N52980 X13.831 Y9.177 
N52990 X13.853 Y9.156 
N53000 X13.874 Y9.135 
N53010 X13.894 Y9.114 
N53020 X13.914 Y9.094 
N53030 X13.933 Y9.075 
N53040 X13.952 Y9.056 
N53050 X13.97 Y9.038 
N53060 X13.987 Y9.021 
N53070 X14.004 Y9.004 
N53080 X14.02 Y8.988 
N53090 X14.036 Y8.972 
N53100 X14.051 Y8.957 
N53110 X14.065 Y8.943 
N53120 X14.079 Y8.929 
N53130 X14.092 Y8.916 
N53140 X14.104 Y8.904 
N53150 X14.116 Y8.892 
N53160 X14.127 Y8.881 
N53170 X14.137 Y8.871 
N53180 X14.147 Y8.861 
N53190 X14.156 Y8.853 
N53200 X14.164 Y8.844 
N53210 X14.171 Y8.837 
N53220 X14.178 Y8.83 
N53230 X14.184 Y8.825 
N53240 X14.189 Y8.819 
N53250 X14.193 Y8.815 
N53260 X14.197 Y8.811 
N53270 X14.199 Y8.809 
N53280 X14.201 Y8.807 
N53290 X14.203 Y8.805 
N53300 X14.204 Y8.805 
N53310 X14.207 
N53320 X14.214 
N53330 X14.217 
N53340 X14.218 
N53350 X14.218 Y8.804 
N53360 Y8.802 
N53370 Y8.798 
N53380 Y8.793 
N53390 Y8.786 
N53400 Y8.778 
N53410 Y8.769 
N53420 Y8.757 
N53430 Y8.745 
N53440 Y8.731 
N53450 Y8.716 
N53460 Y8.699 
N53470 Y8.681 
N53480 Y8.662 
N53490 Y8.641 
N53500 Y8.619 
N53510 Y8.596 
N53520 Y8.571 
N53530 Y8.545 
N53540 Y8.518 
N53550 Y8.49 
N53560 Y8.46 
N53570 Y8.43 
N53580 Y8.398 
N53590 Y8.365 
N53600 Y8.33 
N53610 Y8.295 
N53620 Y8.259 
N53630 Y8.221 
N53640 Y8.182 
N53650 Y8.143 
N53660 Y8.102 
N53670 Y8.06 
N53680 Y8.017 
N53690 Y7.973 
N53700 Y7.928 
N53710 Y7.883 
N53720 Y7.836 
N53730 Y7.788 
N53740 Y7.739 
N53750 Y7.69 
N53760 Y7.639 
N53770 Y7.588 
N53780 Y7.536 
N53790 Y7.483 
N53800 Y7.429 
N53810 Y7.374 
N53820 Y7.319 
N53830 Y7.262 
N53840 Y7.205 
N53850 Y7.147 
N53860 Y7.089 
N53870 Y7.029 
N53880 Y6.969 
N53890 Y6.909 
N53900 Y6.847 
N53910 Y6.785 
N53920 Y6.723 
N53930 Y6.659 
N53940 Y6.595 
N53950 Y6.531 
N53960 Y6.466 
N53970 Y6.4 
N53980 Y6.334 
N53990 Y6.267 
N54000 Y6.132 
N54010 Y5.995 
N54020 Y5.857 
N54030 Y5.716 
N54040 Y5.574 
N54050 Y5.431 
N54060 Y5.286 
N54070 Y5.14 
N54080 Y4.993 
N54090 Y4.845 
N54100 Y4.697 
N54110 Y4.547 
N54120 Y4.247 
N54130 Y3.644 
N54140 Y3.343 
N54150 Y3.194 
N54160 Y3.045 
N54170 Y2.896 
N54180 Y2.749 
N54190 Y2.602 
N54200 Y2.457 
N54210 Y2.313 
N54220 Y2.17 
N54230 Y2.029 
N54240 Y1.889 
N54250 Y1.751 
N54260 Y1.615 
N54270 Y1.481 
N54280 Y1.414 
N54290 Y1.349 
N54300 Y1.283 
N54310 Y1.219 
N54320 Y1.155 
N54330 Y1.091 
N54340 Y1.029 
N54350 Y0.967 
N54360 Y0.905 
N54370 Y0.844 
N54380 Y0.784 
N54390 Y0.725 
N54400 Y0.666 
N54410 Y0.608 
N54420 Y0.551 
N54430 Y0.495 
N54440 Y0.439 
N54450 Y0.384 
N54460 Y0.33 
N54470 Y0.277 
N54480 Y0.224 
N54490 Y0.173 
N54500 Y0.122 
N54510 Y0.073 
N54520 Y0.024 
N54530 Y-0.024 
N54540 Y-0.071 
N54550 Y-0.117 
N54560 Y-0.162 
N54570 Y-0.206 
N54580 Y-0.249 
N54590 Y-0.291 
N54600 Y-0.332 
N54610 Y-0.372 
N54620 Y-0.411 
N54630 Y-0.448 
N54640 Y-0.485 
N54650 Y-0.52 
N54660 Y-0.555 
N54670 Y-0.588 
N54680 Y-0.62 
N54690 Y-0.651 
N54700 Y-0.681 
N54710 Y-0.709 
N54720 Y-0.736 
N54730 Y-0.762 
N54740 Y-0.787 
N54750 Y-0.811 
N54760 Y-0.833 
N54770 Y-0.854 
N54780 Y-0.873 
N54790 Y-0.892 
N54800 Y-0.908 
N54810 Y-0.924 
N54820 Y-0.938 
N54830 Y-0.951 
N54840 Y-0.962 
N54850 Y-0.972 
N54860 Y-0.98 
N54870 Y-0.987 
N54880 Y-0.993 
N54890 Y-0.997 
N54900 Y-0.999 
N54910 Y-1 
N54920 X14.217 Y-1.001 
N54930 X14.216 Y-1.002 
N54940 X14.214 Y-1.004 
N54950 X14.212 Y-1.006 
N54960 X14.209 Y-1.009 
N54970 X14.206 Y-1.012 
N54980 X14.202 Y-1.016 
N54990 X14.198 Y-1.02 
N55000 X14.193 Y-1.025 
N55010 X14.188 Y-1.031 
N55020 X14.182 Y-1.036 
N55030 X14.176 Y-1.042 
N55040 X14.169 Y-1.049 
N55050 X14.162 Y-1.056 
N55060 X14.154 Y-1.064 
N55070 X14.146 Y-1.072 
N55080 X14.138 Y-1.08 
N55090 X14.129 Y-1.089 
N55100 X14.12 Y-1.098 
N55110 X14.11 Y-1.108 
N55120 X14.1 Y-1.118 
N55130 X14.089 Y-1.129 
N55140 X14.078 Y-1.14 
N55150 X14.067 Y-1.151 
N55160 X14.055 Y-1.163 
N55170 X14.043 Y-1.175 
N55180 X14.03 Y-1.188 
N55190 X14.017 Y-1.201 
N55200 X14.004 Y-1.214 
N55210 X13.976 Y-1.242 
N55220 X13.947 Y-1.271 
N55230 X13.916 Y-1.302 
N55240 X13.884 Y-1.334 
N55250 X13.851 Y-1.367 
N55260 X13.817 Y-1.401 
N55270 X13.781 Y-1.437 
N55280 X13.744 Y-1.474 
N55290 X13.706 Y-1.512 
N55300 X13.667 Y-1.551 
N55310 X13.627 Y-1.591 
N55320 X13.586 Y-1.633 
N55330 X13.544 Y-1.675 
N55340 X13.501 Y-1.718 
N55350 X13.457 Y-1.762 
N55360 X13.412 Y-1.806 
N55370 X13.366 Y-1.852 
N55380 X13.32 Y-1.898 
N55390 X13.273 Y-1.945 
N55400 X13.226 Y-1.992 
N55410 X13.178 Y-2.041 
N55420 X13.129 Y-2.089 
N55430 X13.08 Y-2.139 
N55440 X13.03 Y-2.188 
N55450 X12.98 Y-2.238 
N55460 X12.929 Y-2.289 
N55470 X12.827 Y-2.391 
N55480 X12.724 Y-2.494 
N55490 X12.516 Y-2.702 
N55500 X12.412 Y-2.806 
N55510 X12.309 Y-2.91 
N55520 X12.206 Y-3.013 
N55530 X12.104 Y-3.114 
N55540 X12.053 Y-3.165 
N55550 X12.003 Y-3.215 
N55560 X11.954 Y-3.264 
N55570 X11.905 Y-3.313 
N55580 X11.856 Y-3.362 
N55590 X11.808 Y-3.41 
N55600 X11.761 Y-3.457 
N55610 X11.714 Y-3.504 
N55620 X11.668 Y-3.55 
N55630 X11.623 Y-3.595 
N55640 X11.579 Y-3.639 
N55650 X11.535 Y-3.683 
N55660 X11.493 Y-3.726 
N55670 X11.451 Y-3.767 
N55680 X11.41 Y-3.808 
N55690 X11.37 Y-3.848 
N55700 X11.332 Y-3.887 
N55710 X11.294 Y-3.924 
N55720 X11.258 Y-3.961 
N55730 X11.222 Y-3.996 
N55740 X11.188 Y-4.03 
N55750 X11.155 Y-4.063 
N55760 X11.124 Y-4.094 
N55770 X11.094 Y-4.124 
N55780 X11.065 Y-4.153 
N55790 X11.038 Y-4.18 
N55800 X11.025 Y-4.193 
N55810 X11.012 Y-4.206 
N55820 X11 Y-4.218 
N55830 X10.988 Y-4.23 
N55840 X10.977 Y-4.241 
N55850 X10.966 Y-4.252 
N55860 X10.955 Y-4.263 
N55870 X10.945 Y-4.273 
N55880 X10.935 Y-4.283 
N55890 X10.925 Y-4.293 
N55900 X10.916 Y-4.302 
N55910 X10.908 Y-4.31 
N55920 X10.9 Y-4.318 
N55930 X10.892 Y-4.326 
N55940 X10.885 Y-4.333 
N55950 X10.878 Y-4.34 
N55960 X10.872 Y-4.346 
N55970 X10.866 Y-4.352 
N55980 X10.861 Y-4.358 
N55990 X10.856 Y-4.363 
N56000 X10.851 Y-4.367 
N56010 X10.847 Y-4.371 
N56020 X10.844 Y-4.374 
N56030 X10.841 Y-4.377 
N56040 X10.839 Y-4.38 
N56050 X10.837 Y-4.382 
N56060 X10.835 Y-4.383 
N56070 X10.834 Y-4.384 
N56080 X10.834 Y-4.385 
N56090 X10.835 Y-4.386 
N56100 X10.836 Y-4.392 
N56110 X10.84 Y-4.402 
N56120 X10.852 Y-4.445 
N56130 X10.864 Y-4.488 
N56140 X10.875 Y-4.531 
N56150 X10.885 Y-4.574 
N56160 X10.894 Y-4.618 
N56170 X10.902 Y-4.661 
N56180 X10.909 Y-4.705 
N56190 X10.915 Y-4.749 
N56200 X10.919 Y-4.794 
N56210 X10.922 Y-4.839 
N56220 X10.924 Y-4.885 
N56230 X10.925 Y-4.908 
N56240 X10.925 Y-4.92 
N56250 X10.925 Y-4.921 
N56260 X10.925 Y-4.925 
N56270 X10.925 Y-4.932 
N56280 X10.924 Y-4.946 
N56290 X10.924 Y-4.975 
N56300 X10.921 Y-5.032 
N56310 X10.916 Y-5.089 
N56320 X10.91 Y-5.144 
N56330 X10.902 Y-5.2 
N56340 X10.892 Y-5.255 
N56350 X10.88 Y-5.309 
N56360 X10.866 Y-5.362 
N56370 X10.851 Y-5.415 
N56380 X10.834 Y-5.467 
N56390 X10.816 Y-5.519 
N56400 X10.796 Y-5.569 
N56410 X10.774 Y-5.619 
N56420 X10.751 Y-5.668 
N56430 X10.726 Y-5.716 
N56440 X10.7 Y-5.763 
N56450 X10.673 Y-5.81 
N56460 X10.644 Y-5.855 
N56470 X10.614 Y-5.899 
N56480 X10.582 Y-5.943 
N56490 X10.549 Y-5.985 
N56500 X10.515 Y-6.026 
N56510 X10.479 Y-6.066 
N56520 X10.442 Y-6.105 
N56530 X10.404 Y-6.143 
N56540 X10.365 Y-6.18 
N56550 X10.325 Y-6.215 
N56560 X10.284 Y-6.249 
N56570 X10.241 Y-6.282 
N56580 X10.198 Y-6.313 
N56590 X10.153 Y-6.343 
N56600 X10.108 Y-6.372 
N56610 X10.061 Y-6.4 
N56620 X10.014 Y-6.425 
N56630 X9.966 Y-6.45 
N56640 X9.917 Y-6.473 
N56650 X9.867 Y-6.494 
N56660 X9.816 Y-6.514 
N56670 X9.764 Y-6.532 
N56680 X9.712 Y-6.549 
N56690 X9.659 Y-6.564 
N56700 X9.606 Y-6.577 
N56710 X9.551 Y-6.589 
N56720 X9.497 Y-6.598 
N56730 X9.441 Y-6.606 
N56740 X9.385 Y-6.613 
N56750 X9.329 Y-6.617 
N56760 X9.272 Y-6.619 
N56770 X9.214 Y-6.62 
N56780 X9.157 Y-6.619 
N56790 X9.1 Y-6.616 
N56800 X9.044 Y-6.61 
N56810 X8.988 Y-6.604 
N56820 X8.933 Y-6.595 
N56830 X8.878 Y-6.584 
N56840 X8.824 Y-6.572 
N56850 X8.771 Y-6.558 
N56860 X8.718 Y-6.543 
N56870 X8.666 Y-6.525 
N56880 X8.615 Y-6.507 
N56890 X8.564 Y-6.486 
N56900 X8.515 Y-6.464 
N56910 X8.466 Y-6.441 
N56920 X8.418 Y-6.416 
N56930 X8.371 Y-6.389 
N56940 X8.325 Y-6.361 
N56950 X8.28 Y-6.332 
N56960 X8.236 Y-6.301 
N56970 X8.193 Y-6.269 
N56980 X8.151 Y-6.236 
N56990 X8.11 Y-6.202 
N57000 X8.07 Y-6.166 
N57010 X8.031 Y-6.129 
N57020 X7.994 Y-6.09 
N57030 X7.957 Y-6.051 
N57040 X7.922 Y-6.011 
N57050 X7.889 Y-5.969 
N57060 X7.856 Y-5.926 
N57070 X7.825 Y-5.883 
N57080 X7.795 Y-5.838 
N57090 X7.767 Y-5.792 
N57100 X7.74 Y-5.745 
N57110 X7.714 Y-5.698 
N57120 X7.69 Y-5.649 
N57130 X7.667 Y-5.6 
N57140 X7.646 Y-5.55 
N57150 X7.627 Y-5.499 
N57160 X7.609 Y-5.447 
N57170 X7.593 Y-5.395 
N57180 X7.578 Y-5.342 
N57190 X7.566 Y-5.288 
N57200 X7.554 Y-5.234 
N57210 X7.545 Y-5.179 
N57220 X7.537 Y-5.123 
N57230 X7.532 Y-5.067 
N57240 X7.528 Y-5.01 
N57250 X7.526 Y-4.953 
N57260 X7.526 Y-4.896 
N57270 X7.527 Y-4.839 
N57280 X7.531 Y-4.782 
N57290 X7.537 Y-4.726 
N57300 X7.544 Y-4.67 
N57310 X7.553 Y-4.615 
N57320 X7.564 Y-4.56 
N57330 X7.576 Y-4.507 
N57340 X7.591 Y-4.453 
N57350 X7.607 Y-4.401 
N57360 X7.624 Y-4.349 
N57370 X7.644 Y-4.298 
N57380 X7.664 Y-4.248 
N57390 X7.687 Y-4.198 
N57400 X7.711 Y-4.15 
N57410 X7.736 Y-4.102 
N57420 X7.763 Y-4.055 
N57430 X7.791 Y-4.01 
N57440 X7.821 Y-3.965 
N57450 X7.852 Y-3.921 
N57460 X7.884 Y-3.878 
N57470 X7.917 Y-3.836 
N57480 X7.952 Y-3.796 
N57490 X7.988 Y-3.756 
N57500 X8.026 Y-3.718 
N57510 X8.064 Y-3.68 
N57520 X8.104 Y-3.644 
N57530 X8.145 Y-3.61 
N57540 X8.187 Y-3.576 
N57550 X8.23 Y-3.544 
N57560 X8.274 Y-3.513 
N57570 X8.318 Y-3.484 
N57580 X8.364 Y-3.455 
N57590 X8.411 Y-3.429 
N57600 X8.459 Y-3.404 
N57610 X8.508 Y-3.38 
N57620 X8.557 Y-3.358 
N57630 X8.607 Y-3.337 
N57640 X8.659 Y-3.318 
N57650 X8.71 Y-3.301 
N57660 X8.763 Y-3.285 
N57670 X8.816 Y-3.271 
N57680 X8.87 Y-3.258 
N57690 X8.925 Y-3.247 
N57700 X8.98 Y-3.238 
N57710 X9.036 Y-3.231 
N57720 X9.092 Y-3.226 
N57730 X9.149 Y-3.223 
N57740 X9.206 Y-3.221 
N57750 X9.22 Y-3.221 
N57760 X9.224 Y-3.221 
N57770 X9.225 Y-3.221 
N57780 X9.226 
N57790 X9.227 Y-3.221 
N57800 X9.233 Y-3.221 
N57810 X9.256 Y-3.221 
N57820 X9.302 Y-3.223 
N57830 X9.348 Y-3.226 
N57840 X9.393 Y-3.23 
N57850 X9.438 Y-3.236 
N57860 X9.483 Y-3.243 
N57870 X9.527 Y-3.251 
N57880 X9.571 Y-3.26 
N57890 X9.614 Y-3.27 
N57900 X9.656 Y-3.281 
N57910 X9.698 Y-3.292 
N57920 X9.74 Y-3.305 
N57930 X9.76 Y-3.311 
N57940 X9.761 Y-3.311 
N57950 X9.762 Y-3.311 
N57960 X9.763 Y-3.31 
N57970 X9.764 Y-3.308 
N57980 X9.766 Y-3.307 
N57990 X9.769 Y-3.304 
N58000 X9.771 Y-3.302 
N58010 X9.774 Y-3.298 
N58020 X9.778 Y-3.295 
N58030 X9.782 Y-3.291 
N58040 X9.787 Y-3.286 
N58050 X9.791 Y-3.281 
N58060 X9.797 Y-3.276 
N58070 X9.802 Y-3.27 
N58080 X9.808 Y-3.264 
N58090 X9.815 Y-3.258 
N58100 X9.822 Y-3.251 
N58110 X9.829 Y-3.244 
N58120 X9.837 Y-3.236 
N58130 X9.845 Y-3.228 
N58140 X9.862 Y-3.211 
N58150 X9.88 Y-3.193 
N58160 X9.9 Y-3.173 
N58170 X9.921 Y-3.151 
N58180 X9.944 Y-3.129 
N58190 X9.968 Y-3.105 
N58200 X9.993 Y-3.08 
N58210 X10.02 Y-3.053 
N58220 X10.047 Y-3.026 
N58230 X10.076 Y-2.997 
N58240 X10.106 Y-2.967 
N58250 X10.137 Y-2.936 
N58260 X10.168 Y-2.904 
N58270 X10.201 Y-2.872 
N58280 X10.235 Y-2.838 
N58290 X10.27 Y-2.803 
N58300 X10.305 Y-2.767 
N58310 X10.342 Y-2.731 
N58320 X10.379 Y-2.694 
N58330 X10.417 Y-2.656 
N58340 X10.456 Y-2.617 
N58350 X10.495 Y-2.578 
N58360 X10.535 Y-2.537 
N58370 X10.576 Y-2.497 
N58380 X10.617 Y-2.456 
N58390 X10.659 Y-2.414 
N58400 X10.701 Y-2.372 
N58410 X10.744 Y-2.329 
N58420 X10.787 Y-2.286 
N58430 X10.831 Y-2.242 
N58440 X10.919 Y-2.154 
N58450 X11.008 Y-2.065 
N58460 X11.097 Y-1.975 
N58470 X11.188 Y-1.885 
N58480 X11.368 Y-1.705 
N58490 X11.458 Y-1.615 
N58500 X11.547 Y-1.526 
N58510 X11.635 Y-1.438 
N58520 X11.678 Y-1.395 
N58530 X11.721 Y-1.351 
N58540 X11.764 Y-1.309 
N58550 X11.806 Y-1.267 
N58560 X11.848 Y-1.225 
N58570 X11.889 Y-1.184 
N58580 X11.93 Y-1.143 
N58590 X11.97 Y-1.103 
N58600 X12.009 Y-1.064 
N58610 X12.048 Y-1.025 
N58620 X12.086 Y-0.987 
N58630 X12.123 Y-0.95 
N58640 X12.159 Y-0.914 
N58650 X12.195 Y-0.878 
N58660 X12.229 Y-0.843 
N58670 X12.263 Y-0.81 
N58680 X12.296 Y-0.777 
N58690 X12.328 Y-0.745 
N58700 X12.358 Y-0.714 
N58710 X12.388 Y-0.685 
N58720 X12.417 Y-0.656 
N58730 X12.444 Y-0.629 
N58740 X12.471 Y-0.602 
N58750 X12.496 Y-0.577 
N58760 X12.519 Y-0.553 
N58770 X12.542 Y-0.531 
N58780 X12.563 Y-0.51 
N58790 X12.583 Y-0.49 
N58800 X12.601 Y-0.472 
N58810 X12.618 Y-0.455 
N58820 X12.626 Y-0.447 
N58830 X12.634 Y-0.439 
N58840 X12.641 Y-0.432 
N58850 X12.648 Y-0.425 
N58860 X12.654 Y-0.419 
N58870 X12.66 Y-0.413 
N58880 X12.666 Y-0.407 
N58890 X12.671 Y-0.402 
N58900 X12.676 Y-0.397 
N58910 X12.68 Y-0.393 
N58920 X12.684 Y-0.389 
N58930 X12.687 Y-0.385 
N58940 X12.69 Y-0.382 
N58950 X12.693 Y-0.38 
N58960 X12.695 Y-0.377 
N58970 X12.697 Y-0.376 
N58980 X12.699 Y-0.374 
N58990 X12.699 Y-0.373 
N59000 X12.7 Y-0.373 
N59010 Y-0.371 
N59020 Y-0.369 
N59030 Y-0.364 
N59040 Y-0.359 
N59050 Y-0.352 
N59060 Y-0.344 
N59070 Y-0.335 
N59080 Y-0.325 
N59090 Y-0.313 
N59100 Y-0.3 
N59110 Y-0.286 
N59120 Y-0.271 
N59130 Y-0.254 
N59140 Y-0.237 
N59150 Y-0.218 
N59160 Y-0.198 
N59170 Y-0.177 
N59180 Y-0.155 
N59190 Y-0.132 
N59200 Y-0.107 
N59210 Y-0.082 
N59220 Y-0.056 
N59230 Y-0.028 
N59240 Y0 
N59250 Y0.03 
N59260 Y0.06 
N59270 Y0.092 
N59280 Y0.124 
N59290 Y0.158 
N59300 Y0.192 
N59310 Y0.227 
N59320 Y0.263 
N59330 Y0.3 
N59340 Y0.338 
N59350 Y0.377 
N59360 Y0.417 
N59370 Y0.457 
N59380 Y0.499 
N59390 Y0.541 
N59400 Y0.584 
N59410 Y0.628 
N59420 Y0.672 
N59430 Y0.717 
N59440 Y0.764 
N59450 Y0.81 
N59460 Y0.858 
N59470 Y0.906 
N59480 Y0.955 
N59490 Y1.004 
N59500 Y1.055 
N59510 Y1.106 
N59520 Y1.157 
N59530 Y1.209 
N59540 Y1.262 
N59550 Y1.315 
N59560 Y1.369 
N59570 Y1.424 
N59580 Y1.479 
N59590 Y1.534 
N59600 Y1.591 
N59610 Y1.704 
N59620 Y1.82 
N59630 Y1.937 
N59640 Y2.057 
N59650 Y2.177 
N59660 Y2.3 
N59670 Y2.424 
N59680 Y2.548 
N59690 Y2.675 
N59700 Y2.802 
N59710 Y2.93 
N59720 Y3.059 
N59730 Y3.188 
N59740 Y3.319 
N59750 Y3.581 
N59760 Y4.107 
N59770 Y4.369 
N59780 Y4.63 
N59790 Y4.76 
N59800 Y4.889 
N59810 Y5.017 
N59820 Y5.144 
N59830 Y5.27 
N59840 Y5.395 
N59850 Y5.519 
N59860 Y5.641 
N59870 Y5.762 
N59880 Y5.881 
N59890 Y5.998 
N59900 Y6.114 
N59910 Y6.227 
N59920 Y6.284 
N59930 Y6.339 
N59940 Y6.394 
N59950 Y6.449 
N59960 Y6.502 
N59970 Y6.556 
N59980 Y6.608 
N59990 Y6.66 
N60000 Y6.712 
N60010 Y6.763 
N60020 Y6.813 
N60030 Y6.862 
N60040 Y6.911 
N60050 Y6.959 
N60060 Y7.007 
N60070 Y7.054 
N60080 Y7.099 
N60090 Y7.145 
N60100 Y7.189 
N60110 Y7.233 
N60120 Y7.276 
N60130 Y7.318 
N60140 Y7.359 
N60150 Y7.4 
N60160 Y7.439 
N60170 Y7.478 
N60180 Y7.516 
N60190 Y7.553 
N60200 Y7.589 
N60210 Y7.624 
N60220 Y7.658 
N60230 Y7.692 
N60240 Y7.724 
N60250 Y7.755 
N60260 Y7.786 
N60270 Y7.815 
N60280 Y7.844 
N60290 Y7.871 
N60300 Y7.897 
N60310 Y7.922 
N60320 Y7.947 
N60330 Y7.97 
N60340 Y7.992 
N60350 Y8.013 
N60360 Y8.033 
N60370 Y8.051 
N60380 Y8.069 
N60390 Y8.085 
N60400 Y8.1 
N60410 Y8.114 
N60420 Y8.127 
N60430 Y8.139 
N60440 Y8.149 
N60450 Y8.158 
N60460 Y8.166 
N60470 Y8.172 
N60480 Y8.178 
N60490 Y8.182 
N60500 Y8.184 
N60510 Y8.185 
N60520 X12.7 Y8.186 
N60530 X12.699 Y8.186 
N60540 X12.698 Y8.188 
N60550 X12.696 Y8.19 
N60560 X12.693 Y8.192 
N60570 X12.69 Y8.196 
N60580 X12.686 Y8.2 
N60590 X12.681 Y8.204 
N60600 X12.676 Y8.209 
N60610 X12.67 Y8.215 
N60620 X12.664 Y8.222 
N60630 X12.657 Y8.229 
N60640 X12.649 Y8.236 
N60650 X12.641 Y8.245 
N60660 X12.632 Y8.253 
N60670 X12.623 Y8.263 
N60680 X12.613 Y8.273 
N60690 X12.602 Y8.283 
N60700 X12.591 Y8.294 
N60710 X12.58 Y8.306 
N60720 X12.567 Y8.318 
N60730 X12.555 Y8.331 
N60740 X12.541 Y8.344 
N60750 X12.528 Y8.358 
N60760 X12.513 Y8.372 
N60770 X12.499 Y8.387 
N60780 X12.483 Y8.402 
N60790 X12.468 Y8.418 
N60800 X12.451 Y8.434 
N60810 X12.435 Y8.451 
N60820 X12.418 Y8.468 
N60830 X12.4 Y8.486 
N60840 X12.382 Y8.504 
N60850 X12.363 Y8.522 
N60860 X12.344 Y8.541 
N60870 X12.325 Y8.561 
N60880 X12.305 Y8.581 
N60890 X12.285 Y8.601 
N60900 X12.264 Y8.622 
N60910 X12.243 Y8.643 
N60920 X12.221 Y8.664 
N60930 X12.199 Y8.686 
N60940 X12.177 Y8.709 
N60950 X12.154 Y8.731 
N60960 X12.108 Y8.778 
N60970 X12.06 Y8.826 
N60980 X12.01 Y8.875 
N60990 X11.96 Y8.926 
N61000 X11.908 Y8.978 
N61010 X11.855 Y9.031 
N61020 X11.8 Y9.085 
N61030 X11.745 Y9.141 
N61040 X11.688 Y9.197 
N61050 X11.631 Y9.254 
N61060 X11.573 Y9.313 
N61070 X11.513 Y9.372 
N61080 X11.453 Y9.432 
N61090 X11.392 Y9.493 
N61100 X11.33 Y9.555 
N61110 X11.268 Y9.617 
N61120 X11.205 Y9.68 
N61130 X11.142 Y9.744 
N61140 X11.078 Y9.808 
N61150 X11.013 Y9.872 
N61160 X10.949 Y9.937 
N61170 X10.818 Y10.068 
N61180 X10.686 Y10.199 
N61190 X10.555 Y10.331 
N61200 X10.423 Y10.463 
N61210 X10.291 Y10.594 
N61220 X10.161 Y10.725 
N61230 X10.096 Y10.79 
N61240 X10.031 Y10.854 
N61250 X9.967 Y10.918 
N61260 X9.904 Y10.982 
N61270 X9.841 Y11.045 
N61280 X9.779 Y11.107 
N61290 X9.717 Y11.169 
N61300 X9.656 Y11.229 
N61310 X9.596 Y11.29 
N61320 X9.537 Y11.349 
N61330 X9.478 Y11.407 
N61340 X9.421 Y11.465 
N61350 X9.364 Y11.521 
N61360 X9.309 Y11.577 
N61370 X9.254 Y11.631 
N61380 X9.201 Y11.684 
N61390 X9.149 Y11.736 
N61400 X9.099 Y11.787 
N61410 X9.049 Y11.836 
N61420 X9.001 Y11.884 
N61430 X8.955 Y11.931 
N61440 X8.932 Y11.953 
N61450 X8.91 Y11.976 
N61460 X8.888 Y11.998 
N61470 X8.866 Y12.019 
N61480 X8.845 Y12.04 
N61490 X8.825 Y12.061 
N61500 X8.804 Y12.081 
N61510 X8.784 Y12.101 
N61520 X8.765 Y12.121 
N61530 X8.746 Y12.14 
N61540 X8.727 Y12.158 
N61550 X8.709 Y12.176 
N61560 X8.692 Y12.194 
N61570 X8.674 Y12.211 
N61580 X8.658 Y12.228 
N61590 X8.641 Y12.244 
N61600 X8.626 Y12.26 
N61610 X8.61 Y12.275 
N61620 X8.596 Y12.29 
N61630 X8.581 Y12.304 
N61640 X8.568 Y12.318 
N61650 X8.554 Y12.331 
N61660 X8.542 Y12.344 
N61670 X8.53 Y12.356 
N61680 X8.518 Y12.368 
N61690 X8.507 Y12.379 
N61700 X8.496 Y12.389 
N61710 X8.486 Y12.399 
N61720 X8.477 Y12.408 
N61730 X8.468 Y12.417 
N61740 X8.46 Y12.425 
N61750 X8.452 Y12.433 
N61760 X8.445 Y12.44 
N61770 X8.439 Y12.447 
N61780 X8.433 Y12.452 
N61790 X8.428 Y12.458 
N61800 X8.423 Y12.462 
N61810 X8.419 Y12.466 
N61820 X8.416 Y12.469 
N61830 X8.413 Y12.472 
N61840 X8.411 Y12.474 
N61850 X8.41 Y12.475 
N61860 X8.409 Y12.476 
N61870 X8.408 Y12.476 
N61880 X8.407 
N61890 X8.405 
N61900 X8.402 
N61910 X8.399 
N61920 X8.395 
N61930 X8.391 
N61940 X8.386 
N61950 X8.381 
N61960 X8.375 
N61970 X8.368 
N61980 X8.361 
N61990 X8.354 
N62000 X8.345 
N62010 X8.337 
N62020 X8.327 
N62030 X8.318 
N62040 X8.307 
N62050 X8.297 
N62060 X8.285 
N62070 X8.261 
N62080 X8.235 
N62090 X8.206 
N62100 X8.176 
N62110 X8.143 
N62120 X8.109 
N62130 X8.073 
N62140 X8.034 
N62150 X7.994 
N62160 X7.952 
N62170 X7.908 
N62180 X7.863 
N62190 X7.815 
N62200 X7.766 
N62210 X7.715 
N62220 X7.662 
N62230 X7.607 
N62240 X7.551 
N62250 X7.493 
N62260 X7.434 
N62270 X7.373 
N62280 X7.31 
N62290 X7.246 
N62300 X7.18 
N62310 X7.113 
N62320 X7.044 
N62330 X6.974 
N62340 X6.902 
N62350 X6.829 
N62360 X6.754 
N62370 X6.678 
N62380 X6.601 
N62390 X6.523 
N62400 X6.443 
N62410 X6.362 
N62420 X6.279 
N62430 X6.196 
N62440 X6.111 
N62450 X6.025 
N62460 X5.938 
N62470 X5.849 
N62480 X5.76 
N62490 X5.67 
N62500 X5.578 
N62510 X5.485 
N62520 X5.392 
N62530 X5.297 
N62540 X5.202 
N62550 X5.105 
N62560 X5.008 
N62570 X4.91 
N62580 X4.811 
N62590 X4.711 
N62600 X4.61 
N62610 X4.508 
N62620 X4.406 
N62630 X4.303 
N62640 X4.199 
N62650 X4.094 
N62660 X3.989 
N62670 X3.883 
N62680 X3.777 
N62690 X3.67 
N62700 X3.562 
N62710 X3.454 
N62720 X3.345 
N62730 X3.126 
N62740 X2.905 
N62750 X2.683 
N62760 X2.459 
N62770 X2.234 
N62780 X2.008 
N62790 X1.78 
N62800 X1.324 
N62810 X0.41 
N62820 X0.183 
N62830 X-0.044 
N62840 X-0.271 
N62850 X-0.496 
N62860 X-0.72 
N62870 X-0.942 
N62880 X-1.163 
N62890 X-1.382 
N62900 X-1.491 
N62910 X-1.599 
N62920 X-1.707 
N62930 X-1.814 
N62940 X-1.921 
N62950 X-2.027 
N62960 X-2.132 
N62970 X-2.237 
N62980 X-2.341 
N62990 X-2.444 
N63000 X-2.546 
N63010 X-2.648 
N63020 X-2.749 
N63030 X-2.849 
N63040 X-2.948 
N63050 X-3.046 
N63060 X-3.144 
N63070 X-3.24 
N63080 X-3.336 
N63090 X-3.431 
N63100 X-3.524 
N63110 X-3.617 
N63120 X-3.709 
N63130 X-3.799 
N63140 X-3.889 
N63150 X-3.977 
N63160 X-4.064 
N63170 X-4.15 
N63180 X-4.235 
N63190 X-4.319 
N63200 X-4.402 
N63210 X-4.483 
N63220 X-4.563 
N63230 X-4.641 
N63240 X-4.719 
N63250 X-4.795 
N63260 X-4.869 
N63270 X-4.943 
N63280 X-5.015 
N63290 X-5.085 
N63300 X-5.154 
N63310 X-5.221 
N63320 X-5.287 
N63330 X-5.352 
N63340 X-5.414 
N63350 X-5.476 
N63360 X-5.535 
N63370 X-5.593 
N63380 X-5.65 
N63390 X-5.704 
N63400 X-5.757 
N63410 X-5.809 
N63420 X-5.858 
N63430 X-5.906 
N63440 X-5.952 
N63450 X-5.996 
N63460 X-6.038 
N63470 X-6.078 
N63480 X-6.117 
N63490 X-6.153 
N63500 X-6.188 
N63510 X-6.22 
N63520 X-6.251 
N63530 X-6.28 
N63540 X-6.306 
N63550 X-6.331 
N63560 X-6.342 
N63570 X-6.353 
N63580 X-6.363 
N63590 X-6.373 
N63600 X-6.383 
N63610 X-6.391 
N63620 X-6.4 
N63630 X-6.407 
N63640 X-6.415 
N63650 X-6.421 
N63660 X-6.427 
N63670 X-6.433 
N63680 X-6.438 
N63690 X-6.442 
N63700 X-6.446 
N63710 X-6.449 
N63720 X-6.452 
N63730 X-6.454 
N63740 X-6.456 
N63750 X-6.457 
N63760 X-6.459 Y12.474 
N63770 X-6.462 Y12.471 
N63780 X-6.466 Y12.467 
N63790 X-6.472 Y12.461 
N63800 X-6.478 Y12.455 
N63810 X-6.486 Y12.447 
N63820 X-6.495 Y12.438 
N63830 X-6.506 Y12.427 
N63840 X-6.517 Y12.416 
N63850 X-6.53 Y12.403 
N63860 X-6.543 Y12.39 
N63870 X-6.558 Y12.375 
N63880 X-6.573 Y12.359 
N63890 X-6.59 Y12.343 
N63900 X-6.608 Y12.325 
N63910 X-6.626 Y12.306 
N63920 X-6.646 Y12.287 
N63930 X-6.666 Y12.267 
N63940 X-6.687 Y12.245 
N63950 X-6.709 Y12.224 
N63960 X-6.731 Y12.201 
N63970 X-6.755 Y12.177 
N63980 X-6.779 Y12.153 
N63990 X-6.804 Y12.128 
N64000 X-6.83 Y12.102 
N64010 X-6.856 Y12.076 
N64020 X-6.883 Y12.049 
N64030 X-6.91 Y12.022 
N64040 X-6.938 Y11.993 
N64050 X-6.967 Y11.965 
N64060 X-6.996 Y11.936 
N64070 X-7.025 Y11.906 
N64080 X-7.055 Y11.876 
N64090 X-7.085 Y11.846 
N64100 X-7.116 Y11.815 
N64110 X-7.179 Y11.752 
N64120 X-7.243 Y11.688 
N64130 X-7.308 Y11.623 
N64140 X-7.373 Y11.557 
N64150 X-7.439 Y11.49 
N64160 X-7.573 Y11.357 
N64170 X-7.705 Y11.223 
N64180 X-7.771 Y11.157 
N64190 X-7.836 Y11.092 
N64200 X-7.9 Y11.028 
N64210 X-7.963 Y10.965 
N64220 X-7.993 Y10.934 
N64230 X-8.024 Y10.904 
N64240 X-8.054 Y10.874 
N64250 X-8.083 Y10.844 
N64260 X-8.112 Y10.815 
N64270 X-8.141 Y10.786 
N64280 X-8.169 Y10.758 
N64290 X-8.197 Y10.731 
N64300 X-8.223 Y10.704 
N64310 X-8.25 Y10.677 
N64320 X-8.275 Y10.651 
N64330 X-8.3 Y10.626 
N64340 X-8.325 Y10.602 
N64350 X-8.348 Y10.578 
N64360 X-8.371 Y10.556 
N64370 X-8.393 Y10.534 
N64380 X-8.414 Y10.512 
N64390 X-8.434 Y10.492 
N64400 X-8.454 Y10.472 
N64410 X-8.472 Y10.454 
N64420 X-8.49 Y10.436 
N64430 X-8.507 Y10.419 
N64440 X-8.522 Y10.403 
N64450 X-8.537 Y10.389 
N64460 X-8.551 Y10.375 
N64470 X-8.563 Y10.362 
N64480 X-8.575 Y10.351 
N64490 X-8.585 Y10.34 
N64500 X-8.595 Y10.331 
N64510 X-8.603 Y10.323 
N64520 X-8.61 Y10.316 
N64530 X-8.615 Y10.31 
N64540 X-8.62 Y10.306 
N64550 X-8.623 Y10.303 
N64560 X-8.624 Y10.301 
N64570 X-8.625 Y10.301 
N64580 X-8.625 Y10.3 
N64590 X-8.618 Y10.278 
N64600 X-8.606 Y10.236 
N64610 X-8.594 Y10.193 
N64620 X-8.583 Y10.15 
N64630 X-8.573 Y10.107 
N64640 X-8.564 Y10.063 
N64650 X-8.556 Y10.019 
N64660 X-8.55 Y9.975 
N64670 X-8.544 Y9.931 
N64680 X-8.539 Y9.886 
N64690 X-8.536 Y9.841 
N64700 X-8.535 Y9.795 
N64710 X-8.534 Y9.772 
N64720 X-8.534 Y9.766 
N64730 X-8.534 Y9.765 
N64740 Y9.764 
N64750 Y9.763 
N64760 X-8.534 Y9.76 
N64770 X-8.534 Y9.745 
N64780 X-8.536 Y9.688 
N64790 X-8.539 Y9.631 
N64800 X-8.545 Y9.575 
N64810 X-8.552 Y9.519 
N64820 X-8.561 Y9.464 
N64830 X-8.572 Y9.409 
N64840 X-8.584 Y9.356 
N64850 X-8.598 Y9.302 
N64860 X-8.614 Y9.25 
N64870 X-8.631 Y9.198 
N64880 X-8.65 Y9.147 
N64890 X-8.671 Y9.097 
N64900 X-8.693 Y9.047 
N64910 X-8.717 Y8.998 
N64920 X-8.742 Y8.951 
N64930 X-8.769 Y8.904 
N64940 X-8.797 Y8.858 
N64950 X-8.826 Y8.813 
N64960 X-8.857 Y8.769 
N64970 X-8.889 Y8.726 
N64980 X-8.923 Y8.684 
N64990 X-8.958 Y8.643 
N65000 X-8.994 Y8.604 
N65010 X-9.031 Y8.565 
N65020 X-9.069 Y8.528 
N65030 X-9.109 Y8.492 
N65040 X-9.15 Y8.457 
N65050 X-9.191 Y8.423 
N65060 X-9.234 Y8.391 
N65070 X-9.278 Y8.36 
N65080 X-9.323 Y8.33 
N65090 X-9.369 Y8.302 
N65100 X-9.416 Y8.275 
N65110 G00 Z0 
N65120 G00 X0 Y0
*)
